{attribute 'GeneratedUsingTerminal: EL3681-0000-0017'}
{attribute addProperty BoxType "EL3681-0000-0017"}
{attribute addProperty Id "CtrlAT %Q*Ctrl_56BB2DF23"}
{attribute addProperty CRC "923850567"}
{attribute addProperty Size "3"}
TYPE SAI_Range_3710D747 EXTENDS OutputBase_10CEE7DE :
STRUCT
	{attribute addProperty Name "Ctrl"}
	Ctrl AT %Q* : Ctrl_56BB2DF2;
END_STRUCT
END_TYPE

(* stored: Version 1.2.0.0, ProductVersion 3.1.4024.9
   DUT SAI_Range_3710D747: Id {eac275b2-983c-461b-9adb-fa190655e0a7} *)
